# EPICS IOC start-up script: iocsh/ethercatmcAnalogOutput.iocsh
ethercatmcCreateAsynParam $(MOTOR_PORT) $(ASYNPARAMNAME)      Float64
ethercatmcCreateAsynParam $(MOTOR_PORT) $(ASYNPARAMNAME)_DESC Octet

dbLoadRecords("ethercatmcAnalogOutput.template", "P=$(P), R=$(R), MOTOR_PORT=$(MOTOR_PORT), CHNO=$(CHNO), ASYNPARAMNAME=$(ASYNPARAMNAME), PREC=$(PREC), EGU=$(EGU)")
